FUNCTION_BLOCK PercentGinProduct (* Composite Function Block Type *)
  (* Standard: 61499-2 *)
  (* Version 0.0, 2018-10-14, 4DIAC-IDE, 4DIAC-Consortium *)
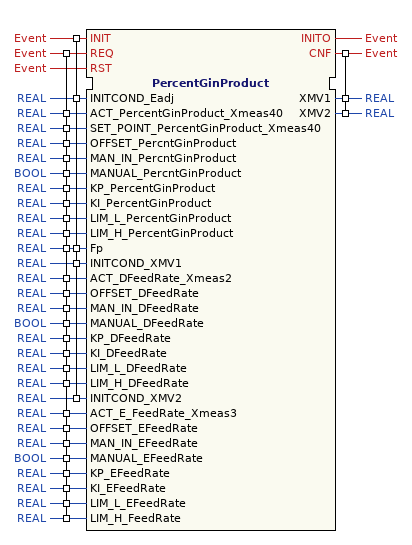
  EVENT_INPUT
    INIT WITH INITCOND_Eadj, INITCOND_XMV1, INITCOND_XMV2, Fp; (* Initialization Request *)
    REQ WITH ACT_PercentGinProduct_Xmeas40, SET_POINT_PercentGinProduct_Xmeas40, OFFSET_PercntGinProduct, MAN_IN_PercntGinProduct, MANUAL_PercntGinProduct, KP_PercentGinProduct, KI_PercentGinProduct, LIM_L_PercentGinProduct, LIM_H_PercentGinProduct, ACT_DFeedRate_Xmeas2, OFFSET_DFeedRate, MAN_IN_DFeedRate, MANUAL_DFeedRate, KP_DFeedRate, KI_DFeedRate, LIM_L_DFeedRate, LIM_H_DFeedRate, ACT_E_FeedRate_Xmeas3, OFFSET_EFeedRate, MAN_IN_EFeedRate, MANUAL_EFeedRate, KP_EFeedRate, KI_EFeedRate, LIM_L_EFeedRate, LIM_H_FeedRate, Fp; (* Normal Execution Request *)
    RST;
  END_EVENT
  EVENT_OUTPUT
    INITO; (* Initialization Confirm *)
    CNF WITH XMV1, XMV2; (* Execution Confirmation *)
  END_EVENT
  VAR_INPUT
    INITCOND_Eadj : REAL;
    ACT_PercentGinProduct_Xmeas40 : REAL;
    SET_POINT_PercentGinProduct_Xmeas40 : REAL;
    OFFSET_PercntGinProduct : REAL;
    MAN_IN_PercntGinProduct : REAL;
    MANUAL_PercntGinProduct : BOOL;
    KP_PercentGinProduct : REAL;
    KI_PercentGinProduct : REAL;
    LIM_L_PercentGinProduct : REAL;
    LIM_H_PercentGinProduct : REAL;
    Fp : REAL;
    INITCOND_XMV1 : REAL;
    ACT_DFeedRate_Xmeas2 : REAL;
    OFFSET_DFeedRate : REAL;
    MAN_IN_DFeedRate : REAL;
    MANUAL_DFeedRate : BOOL;
    KP_DFeedRate : REAL;
    KI_DFeedRate : REAL;
    LIM_L_DFeedRate : REAL;
    LIM_H_DFeedRate : REAL;
    INITCOND_XMV2 : REAL;
    ACT_E_FeedRate_Xmeas3 : REAL;
    OFFSET_EFeedRate : REAL;
    MAN_IN_EFeedRate : REAL;
    MANUAL_EFeedRate : BOOL;
    KP_EFeedRate : REAL;
    KI_EFeedRate : REAL;
    LIM_L_EFeedRate : REAL;
    LIM_H_FeedRate : REAL;
  END_VAR
  VAR_OUTPUT
    XMV1 : REAL;
    XMV2 : REAL;
  END_VAR
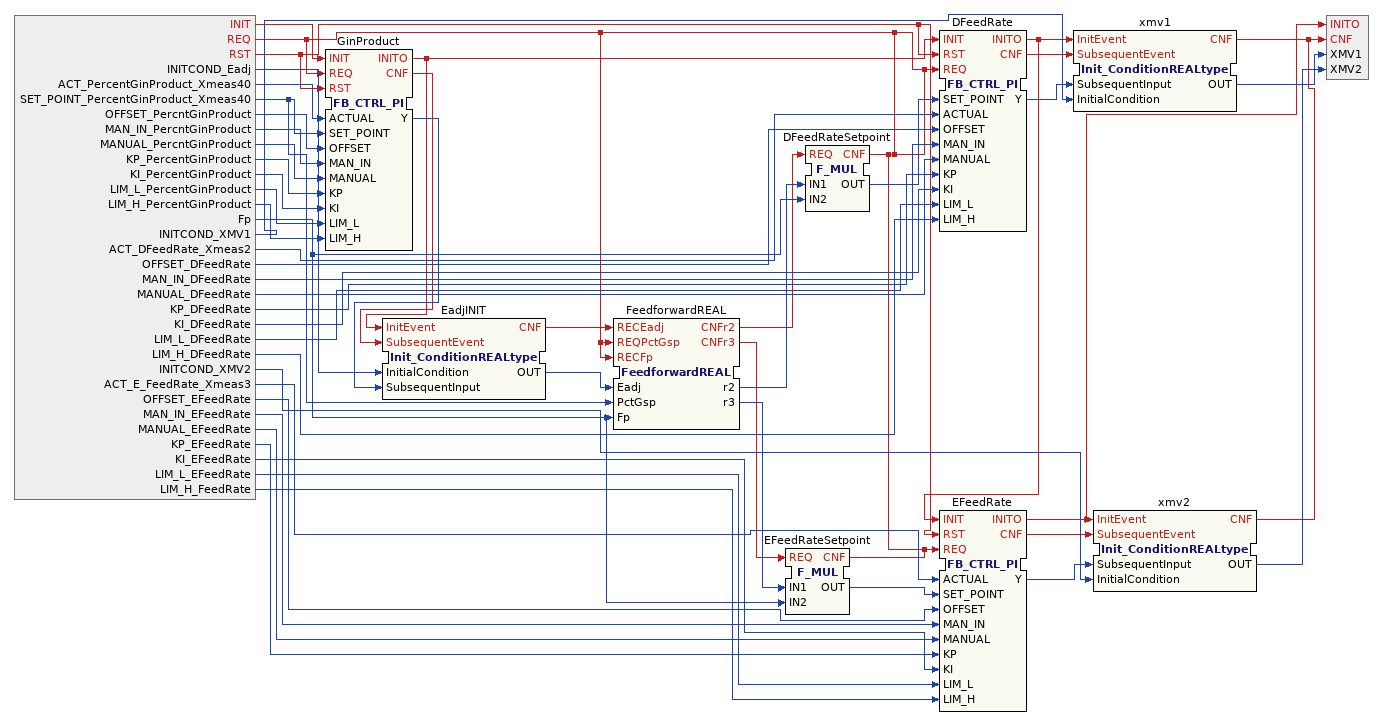
  FBS
    GinProduct : FB_CTRL_PI;
    EadjINIT : Init_ConditionREALtype;
    FeedforwardREAL : FeedforwardREAL;
    DFeedRateSetpoint : F_MUL;
    EFeedRateSetpoint : F_MUL;
    DFeedRate : FB_CTRL_PI;
    EFeedRate : FB_CTRL_PI;
    xmv1 : Init_ConditionREALtype;
    xmv2 : Init_ConditionREALtype;
  END_FBS
  EVENT_CONNECTIONS
    INIT TO GinProduct.INIT;
    GinProduct.INITO TO EadjINIT.InitEvent;
    REQ TO GinProduct.REQ;
    GinProduct.CNF TO EadjINIT.SubsequentEvent;
    GinProduct.INITO TO DFeedRate.INIT;
    DFeedRate.INITO TO xmv1.InitEvent;
    DFeedRate.INITO TO EFeedRate.INIT;
    EFeedRate.INITO TO xmv2.InitEvent;
    RST TO GinProduct.RST;
    RST TO DFeedRate.RST;
    RST TO EFeedRate.RST;
    EadjINIT.CNF TO FeedforwardREAL.RECEadj;
    REQ TO FeedforwardREAL.REQPctGsp;
    FeedforwardREAL.CNFr2 TO DFeedRateSetpoint.REQ;
    DFeedRateSetpoint.CNF TO DFeedRate.REQ;
    REQ TO DFeedRate.REQ;
    DFeedRate.CNF TO xmv1.SubsequentEvent;
    xmv1.CNF TO CNF;
    xmv2.CNF TO CNF;
    EFeedRate.INITO TO INITO;
    FeedforwardREAL.CNFr3 TO EFeedRateSetpoint.REQ;
    EFeedRate.CNF TO xmv2.SubsequentEvent;
    EFeedRateSetpoint.CNF TO EFeedRate.REQ;
    REQ TO EFeedRate.REQ;
    REQ TO FeedforwardREAL.RECFp;
  END_CONNECTIONS
  DATA_CONNECTIONS
    INITCOND_Eadj TO EadjINIT.InitialCondition;
    GinProduct.Y TO EadjINIT.SubsequentInput;
    ACT_PercentGinProduct_Xmeas40 TO GinProduct.ACTUAL;
    SET_POINT_PercentGinProduct_Xmeas40 TO GinProduct.SET_POINT;
    OFFSET_PercntGinProduct TO GinProduct.OFFSET;
    MAN_IN_PercntGinProduct TO GinProduct.MAN_IN;
    MANUAL_PercntGinProduct TO GinProduct.MANUAL;
    KP_PercentGinProduct TO GinProduct.KP;
    KI_PercentGinProduct TO GinProduct.KI;
    LIM_L_PercentGinProduct TO GinProduct.LIM_L;
    LIM_H_PercentGinProduct TO GinProduct.LIM_H;
    EadjINIT.OUT TO FeedforwardREAL.Eadj;
    SET_POINT_PercentGinProduct_Xmeas40 TO FeedforwardREAL.PctGsp;
    Fp TO FeedforwardREAL.Fp;
    FeedforwardREAL.r2 TO DFeedRateSetpoint.IN1;
    DFeedRateSetpoint.OUT TO DFeedRate.SET_POINT;
    DFeedRate.Y TO xmv1.SubsequentInput;
    xmv1.OUT TO XMV1;
    xmv2.OUT TO XMV2;
    EFeedRate.Y TO xmv2.SubsequentInput;
    ACT_DFeedRate_Xmeas2 TO DFeedRate.ACTUAL;
    INITCOND_XMV1 TO xmv1.InitialCondition;
    OFFSET_DFeedRate TO DFeedRate.OFFSET;
    FeedforwardREAL.r3 TO EFeedRateSetpoint.IN1;
    Fp TO EFeedRateSetpoint.IN2;
    Fp TO DFeedRateSetpoint.IN2;
    MAN_IN_DFeedRate TO DFeedRate.MAN_IN;
    MANUAL_DFeedRate TO DFeedRate.MANUAL;
    KP_DFeedRate TO DFeedRate.KP;
    KI_DFeedRate TO DFeedRate.KI;
    LIM_L_DFeedRate TO DFeedRate.LIM_L;
    LIM_H_DFeedRate TO DFeedRate.LIM_H;
    INITCOND_XMV2 TO xmv2.InitialCondition;
    ACT_E_FeedRate_Xmeas3 TO EFeedRate.ACTUAL;
    EFeedRateSetpoint.OUT TO EFeedRate.SET_POINT;
    OFFSET_EFeedRate TO EFeedRate.OFFSET;
    MAN_IN_EFeedRate TO EFeedRate.MAN_IN;
    MANUAL_EFeedRate TO EFeedRate.MANUAL;
    KP_EFeedRate TO EFeedRate.KP;
    KI_EFeedRate TO EFeedRate.KI;
    LIM_L_EFeedRate TO EFeedRate.LIM_L;
    LIM_H_FeedRate TO EFeedRate.LIM_H;
  END_CONNECTIONS
END_FUNCTION_BLOCK
